// TIA Portal V20 export
FUNCTION "ClearAlarms" : Void   // FC14, SCL
{ S7_Optimized_Access := 'TRUE' }
// stored: IsIECCheckEnabled true, SetENOAutomatically true
   VAR_IN_OUT
      error : Array[*] of "LAF_typeAlarm";   // Errors
      warning : Array[*] of "LAF_typeAlarm";   // Warnings
      information : Array[*] of "LAF_typeAlarm";   // Informations of the EM
      criteriaAnalysis : Array[*] of "LAF_typeAlarm";   // CriteriaAnalysis of the EM
   END_VAR
   VAR_TEMP
      tempIndex : DInt;   // For loop variable
   END_VAR
   VAR CONSTANT
      NO_REACTION : USInt;
   END_VAR
BEGIN
   REGION BLOCK INFO HEADER
     //===============================================================================
     // Siemens AG / (c)Copyright 2025
     //-------------------------------------------------------------------------------
     // Title:            LAF_ClearAlarms
     // Comment/Function: Clears all the current active alarms
     // Library/Family:   LAF - Library of Automation Framework
     // Author:           Siemens Digital Industries
     // Tested with:      S7-PLCSIM V20 
     // Engineering:      TIA Portal V20
     // Restrictions:     -
     // Requirements:     -
     //-------------------------------------------------------------------------------
     // Change log table:
     // Version  | Date       | Expert in charge        | Changes applied
     //----------|------------|-------------------------|-----------------------------
     // 01.01.00 | 21.06.2024 | SIMATIC Systems Support | First released version
     // 01.02.00 | 05.08.2024 | SIMATIC Systems Support | Block information properties updated
     // 02.00.00 | 31.03.2025 | SIMATIC Systems Support | Header information updated and removed commandsToUnit
     //===============================================================================
   END_REGION BLOCK INFO HEADER

   REGION errorNoReaction
     FOR #tempIndex := LOWER_BOUND(ARR := #error, DIM := 1) TO UPPER_BOUND(ARR := #error, DIM := 1) DO
       #error[#tempIndex].trigger := false;
     END_FOR;
   END_REGION


   REGION warningNoReaction
     FOR #tempIndex := LOWER_BOUND(ARR := #warning, DIM := 1) TO UPPER_BOUND(ARR := #warning, DIM := 1) DO
       #warning[#tempIndex].trigger := false;
     END_FOR;
   END_REGION


   REGION information
     FOR #tempIndex := LOWER_BOUND(ARR := #information, DIM := 1) TO UPPER_BOUND(ARR := #information, DIM := 1) DO
       #information[#tempIndex].trigger := false;
     END_FOR;
   END_REGION

   REGION criteriaAnalysis
     FOR #tempIndex := LOWER_BOUND(ARR := #criteriaAnalysis, DIM := 1) TO UPPER_BOUND(ARR := #criteriaAnalysis, DIM := 1) DO
       #criteriaAnalysis[#tempIndex].trigger := false;
     END_FOR;
   END_REGION
END_FUNCTION
